# EPICS substitutions: iocs/motorZynqIOC/motorZynqIOCApp/Db/zynqMotor.substitutions
file "db/zynqMotor.template"
{
pattern
{P,      M,                PORT,  ADDR, FULL_STEPS_PER_REV}
{"Det",  "{Sample-Ax:1}",  ZYNQ1, 0, 200}
{"Det",  "{Sample-Ax:2}",  ZYNQ1, 1, 200}
{"Det",  "{Sample-Ax:3}",  ZYNQ1, 2, 200}
{"Det",  "{Sample-Ax:4}",  ZYNQ1, 3, 200}
}
